Yaskawa INFORM job: FECHA_GRAMPOS.JBI

/JOB
//NAME FECHA_GRAMPOS
///FOLDERNAME GRAMPOS
//POS
///NPOS 0,0,0,0,0,0
//INST
///DATE 2022/06/09 09:24
///ATTR SC,RW
NOP
DOUT OT#(537) ON
DOUT OT#(538) OFF
WAIT IN#(538)=ON
WAIT IN#(540)=ON
WAIT IN#(542)=ON
WAIT IN#(544)=ON
END
